FUNCTION_BLOCK FB_ElectricityMeter EXTENDS FB_Sensor
VAR_INPUT
	aElectricityMeterTelegramm	: ARRAY[1..cMBUS_MaxTelegrams] OF ST_MBus_Data2;
END_VAR
VAR_OUTPUT
	fWork : REAL; //Wh
	fPower : REAL; //W
END_VAR
VAR
	{attribute 'OPC.UA.DA' := '1'}
	sensorState : ST_ElectricityMeterState;
END_VAR

sensorState.fWork := STRING_TO_REAL(aElectricityMeterTelegramm[1].arrData[1].sValue);
sensorState.fPower := STRING_TO_REAL(aElectricityMeterTelegramm[1].arrData[2].sValue);

//set outputs
fWork := sensorState.fWork;
fPower := sensorState.fPower;

END_FUNCTION_BLOCK

(* stored: Version 1.1.0.1, ProductVersion 3.1.4024.10
   POU FB_ElectricityMeter: Id {14f8a120-a526-4f46-883e-e3576a0e0d1b}, SpecialFunc None *)
